// TIA Portal V18 export
// export: Created 2025-12-01T17:51:26.5022992Z, ExportSetting None, DisplayName Totally Integrated Automation Portal, DisplayVersion V18 Update 5, DisplayName TIA Portal Openness, DisplayVersion V18 Update 5, DisplayName TIA Portal Teamcenter Gateway, DisplayVersion V18, DisplayName TIA Portal Version Control Interface, DisplayVersion V18, DisplayName STEP 7 Professional, DisplayVersion V18 Update 5, DisplayName STEP 7 Safety, DisplayVersion V18, DisplayName WinCC Professional, DisplayVersion V18 Update 5
DATA_BLOCK "Station2UnLoadData"   // DB513
{ S7_Optimized_Access := 'FALSE' }
// stored: AutoNumber false
   VAR
      "PLC.PartTypeID" : Int;
      "PLC.Station2DMXCode" : String[128];
      "PLC.Station2RecipeNo" : Int;
      "PLC.PartStatus" : Int;
      "PLC.SubPartSN1" : String[128];
      "PLC.TransferTime" : String[128];
      Spare : Byte;
      Spare_1 : Byte;
      Spare_2 : Byte;
      Spare_3 : Byte;
      Spare_4 : Byte;
      Spare_5 : Byte;
      Spare_6 : Byte;
      Spare_7 : Byte;
      Spare_8 : Byte;
      Spare_9 : Byte;
      Spare_10 : Byte;
      "MES.ErrorCode" : Int;
      "MES.ErrorMsg" : String[128];
   END_VAR
BEGIN
END_DATA_BLOCK
